// TIA Portal V21 export
// export: Created 2000-01-01T00:00:00.0000000Z, ExportSetting None
FUNCTION_BLOCK "FB_StartStop"   // FB2, SCL
{ S7_Optimized_Access := 'TRUE' }
// 起保停（Start-Hold-Stop）逻辑：急停优先 > 停止优先 > 启动锁存。
// 当 EStop=TRUE 时立即复位 Run。
// 否则当 Stop=TRUE 时复位 Run。
// 否则当 Start=TRUE 时置位 Run（自保持）。
// stored: SetENOAutomatically false
   VAR_INPUT
      Start : Bool;   // 启动按钮（瞬时上升沿置位 Run）
      Stop : Bool;   // 停止按钮（瞬时复位 Run）
      EStop : Bool;   // 急停（最高优先级，强制复位 Run）
   END_VAR
   VAR_OUTPUT
      Run : Bool;   // 运行输出（起保停锁存位）
   END_VAR
BEGIN
// 起保停核心逻辑
// 急停 > 停止 > 启动 三段优先级 IF/ELSIF
   IF #EStop THEN
     #Run := FALSE;
   ELSIF #Stop THEN
     #Run := FALSE;
   ELSIF #Start THEN
     #Run := TRUE;
   END_IF;
END_FUNCTION_BLOCK
